// TIA Portal V17 export
// export: Created 2022-07-20T07:02:37.7621111Z, ExportSetting WithDefaults, DisplayName Totally Integrated Automation Portal, DisplayVersion V17, DisplayName TIA Portal Openness, DisplayVersion V17, DisplayName TIA Portal Version Control Interface, DisplayVersion V17, DisplayName SINAMICS Startdrive Advanced, DisplayVersion V17, DisplayName SINAMICS Startdrive G130, G150, S120, S150, SINAMICS MV, S210, DisplayVersion V17, DisplayName SINAMICS Startdrive G110M, G120, G120C, G120D, G120P, G115D, DisplayVersion V17, DisplayName STEP 7 Professional, DisplayVersion V17, DisplayName STEP 7 Safety, DisplayVersion V17, DisplayName WinCC Advanced, DisplayVersion V17
VAR_GLOBAL   // PLC tag table "P2WeighScales_TLM8_CommunicationTable"
   P2WeighScales_TLM8_CommandRegister AT %QW0 : UInt;
   P2WeighScales_TLM8_DigitalOutputsCommand AT %QW2 : UInt;
   P2WeighScales_TLM8_WriteExchangeRegister AT %QD4 : UDInt;
   P2WeighScales_TLM8_WeightLoadCell_1 AT %IW0 : Int;
   P2WeighScales_TLM8_WeightLoadCell_2 AT %IW2 : Int;
   P2WeighScales_TLM8_WeightLoadCell_3 AT %IW4 : Int;
   P2WeighScales_TLM8_WeightLoadCell_4 AT %IW6 : Int;
   P2WeighScales_TLM8_WeightLoadCell_5 AT %IW8 : Int;
   P2WeighScales_TLM8_WeightLoadCell_6 AT %IW10 : Int;
   P2WeighScales_TLM8_WeightLoadCell_7 AT %IW12 : Word;
   P2WeighScales_TLM8_WeightLoadCell_8 AT %IW14 : Int;
   P2WeighScales_TLM8_StatusRegister AT %IW16 : UInt;
END_VAR
